(* CODESYS project Uppgift 6.project

Project tree, tasks and I/O mapping:
  Device : CODESYS Control Win V3, 3S - Smart Software Solutions GmbH, order no. 305021, version 3.5.10.40
    application Application
      libraries: Standard, * (System)
      task MainTask (cyclic, interval t#20ms, priority 1) calls PLC_PRG
      program PLC_PRG [LD]
      global variables GVL
*)

// Device/Application/GVL
{attribute 'qualified_only'}
VAR_GLOBAL
	Motor_fwr: BOOL;
	Sensor_b: BOOL;
	Sensor_a: BOOL;
END_VAR

// Device/Application/PLC_PRG
PROGRAM PLC_PRG
VAR
	Motor_fwr: BOOL;
	Sensor_b: BOOL;
	Sensor_a: BOOL;
END_VAR

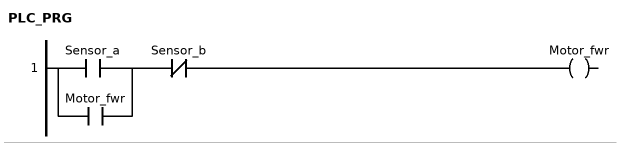
// NETWORK 1
Motor_fwr := (Sensor_a OR Motor_fwr) AND NOT Sensor_b;

END_PROGRAM
